{attribute addProperty BoxType "EL3314-0010-0016"}
{attribute addProperty Id "UnderrangeBIT10.1251OverrangeBIT10.1252ErrorBIT10.1257TxPDO_StateBIT10.12515TxPDO_ToggleBIT10.1259"}
{attribute addProperty CRC "4145063443"}
{attribute addProperty SizeInBites "93"}
{attribute addProperty SizeInBytes "11.625"}
{warning 'Size of this structure is not a multiple of 8 bits!!!'}
TYPE Status_F710A613 :
STRUCT
	{attribute addProperty Name "Underrange"}
	Underrange : BIT;
	{attribute addProperty Name "Overrange"}
	Overrange : BIT;
	{attribute 'hide'}
	reserve_1_BOOL_0 : BOOL;
	{attribute 'hide'}
	reserve_1_BOOL_1 : BOOL;
	{attribute 'hide'}
	reserve_1_BOOL_2 : BOOL;
	{attribute 'hide'}
	reserve_1_BOOL_3 : BOOL;
	{attribute addProperty Name "Error"}
	Error : BIT;
	{attribute 'hide'}
	reserve_2_BOOL_0 : BOOL;
	{attribute 'hide'}
	reserve_2_BOOL_1 : BOOL;
	{attribute 'hide'}
	reserve_2_BOOL_2 : BOOL;
	{attribute 'hide'}
	reserve_2_BOOL_3 : BOOL;
	{attribute 'hide'}
	reserve_2_BOOL_4 : BOOL;
	{attribute 'hide'}
	reserve_2_BOOL_5 : BOOL;
	{attribute 'hide'}
	reserve_2_BOOL_6 : BOOL;
	{attribute addProperty Name "TxPDO_State"}
	TxPDO_State : BIT;
	{attribute addProperty Name "TxPDO_Toggle"}
	TxPDO_Toggle : BIT;
END_STRUCT
END_TYPE

(* stored: Version 1.2.0.0, ProductVersion 3.1.4024.9
   DUT Status_F710A613: Id {6842753d-13a5-4a20-b7eb-0cc0c94899a1} *)
